FUNCTION_BLOCK FB_TestSuiteExtendedHE_SATT EXTENDS FB_TestSuiteExtended
VAR
END_VAR

END_FUNCTION_BLOCK

(* stored: Version 1.1.0.1
   POU FB_TestSuiteExtendedHE_SATT: Id {c7452345-6edb-4c90-a4bd-7ac47252e955}, SpecialFunc None *)
